// TIA Portal V18 export
// export: Created 2026-03-12T16:04:35.2484004Z, ExportSetting WithDefaults, DisplayName Totally Integrated Automation Portal, DisplayVersion V18 Update 5, DisplayName TIA Portal Openness, DisplayVersion V18 Update 5, DisplayName TIA Portal Version Control Interface, DisplayVersion V18, DisplayName SINAMICS Startdrive Advanced, DisplayVersion V18, DisplayName SINAMICS Startdrive G130, G150, S120, S150, SINAMICS MV, S210, DisplayVersion V18, DisplayName SINAMICS Startdrive G110M, G120, G120C, G120D, G120P, G115D, DisplayVersion V18, DisplayName STEP 7 Professional, DisplayVersion V18 Update 5, DisplayName STEP 7 Safety, DisplayVersion V18, DisplayName WinCC Professional, DisplayVersion V18 Update 5
FUNCTION_BLOCK "FB ALARME DIGITAL"   // FB3, LAD
TITLE = Function Block ALARME DIGITAL
{ S7_Optimized_Access := 'TRUE' }
VERSION : 0.1
// Tratamento de alarmes: Setando e Resetando sinais digitais relacionados aos alarmes
// stored: AutoNumber true, IsIECCheckEnabled false, IsRetainMemResEnabled false, MemoryReserve 100, SetENOAutomatically false, UDAEnableTagReadback false
   VAR_INPUT
      SINAL_ENTRADA_DIGITAL : Bool;   // Entrada digital do sinal elétrico
   END_VAR
   VAR_OUTPUT
      BD_GLOBAL_ALARME : Bool;   // Saída digital instanciada no FB
   END_VAR
   VAR
      RESET_TIME : IEC_TIMER;   // Reset do alarme caso o sinal seja interrompido
      ACIONA_BD_ALARME : Bool;   // Chaveamento para acionar/desacionar o alarme
   END_VAR
BEGIN

REGION Network 1: SET RESET
   // Recebendo sinal da I/O do equipamento e setando o alarme dentro da DB. Após a entrada identificar nível baixo (0) a saída do alarme é resetada conforme tempo configurado.
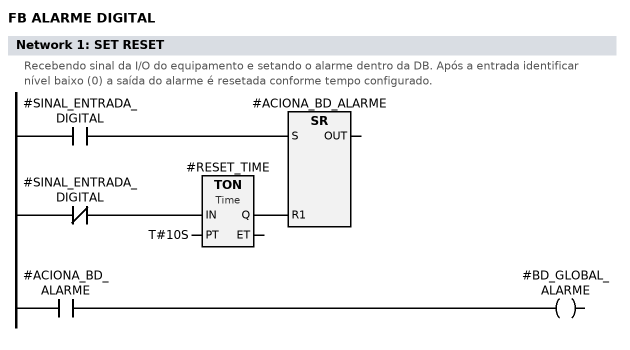
   RUNG wire#powerrail
      Contact( #SINAL_ENTRADA_DIGITAL )
      S_SR(operand := #ACIONA_BD_ALARME, r1 := wire#w1)
   END_RUNG
   RUNG wire#powerrail
      I_Contact( #SINAL_ENTRADA_DIGITAL )
      { S7_Templates := "time_type := Time" } #RESET_TIME.TON(pt := T#10S, et =>)
   END_RUNG wire#w1
   RUNG wire#powerrail
      Contact( #ACIONA_BD_ALARME )
      Coil( #BD_GLOBAL_ALARME )
   END_RUNG
   // the same network as SCL:
   #RESET_TIME.TON(IN := NOT #SINAL_ENTRADA_DIGITAL, PT := T#10S);
   IF #SINAL_ENTRADA_DIGITAL THEN
       #ACIONA_BD_ALARME := TRUE;   // SR flip-flop
   END_IF;
   IF #RESET_TIME.Q THEN #ACIONA_BD_ALARME := FALSE; END_IF;
   #BD_GLOBAL_ALARME := #ACIONA_BD_ALARME;
END_REGION
END_FUNCTION_BLOCK
